INTERFACE I_Dictionary EXTENDS I_KeyValueCollection

METHOD PUBLIC AddOrUpdate
VAR_INPUT
	Key : T_MAXSTRING;
	Value : ANY;
END_VAR
END_METHOD

METHOD PUBLIC Clear
VAR_INPUT
END_VAR
END_METHOD

METHOD PUBLIC ContainsKey : BOOL
VAR_INPUT
	Key : T_MAXSTRING;
END_VAR
END_METHOD

METHOD PUBLIC GetKeys : I_Collection
END_METHOD

METHOD PUBLIC Remove
VAR_INPUT
	Key : T_MAXSTRING;
END_VAR
END_METHOD

METHOD PUBLIC TryAdd : BOOL
VAR_INPUT
	Key : T_MAXSTRING;
	Value : ANY;
END_VAR
END_METHOD

METHOD PUBLIC TryGetValue : BOOL
VAR_INPUT
	Key : T_MAXSTRING;
	Destination	: ANY;
END_VAR
END_METHOD

METHOD PUBLIC TryGetValueTo : BOOL
VAR_INPUT
	Key : T_MAXSTRING;
	DestinationAddress : PVOID;
	DestinationSize : UDINT;
END_VAR
END_METHOD

END_INTERFACE

(* stored: Version 1.1.0.1, ProductVersion 3.1.4024.12
   Itf I_Dictionary: Id {06f7de23-27cf-4103-9cac-bc3822cddc82}
   Method AddOrUpdate: Id {641eaa0a-e872-4d4b-bc8a-d398207c70c2}
   Method Clear: Id {7bb7b21a-499d-4c0e-8c5c-4ea2106057a5}
   Method ContainsKey: Id {ffccb942-d8e8-4e6d-bd12-715818c73d38}
   Method GetKeys: Id {8c2ec7fd-25f6-48b1-9d92-32f03d6814c3}
   Method Remove: Id {9cbd6d40-ae4d-429a-8f44-1c26ba8dd518}
   Method TryAdd: Id {d7a05a01-800c-4d04-a211-24735d139ae7}
   Method TryGetValue: Id {b6af0a3f-85a9-4af8-8c8a-adb57519096b}
   Method TryGetValueTo: Id {d6adcfe3-d192-411f-8625-ea56b0400ab0} *)
